INTERFACE I_UnitTest EXTENDS __SYSTEM.IQueryInterface

METHOD InitBase
VAR_INPUT
END_VAR
END_METHOD

PROPERTY Name : T_MaxString
GET
END_GET
END_PROPERTY

METHOD FINAL RunTest
END_METHOD

PROPERTY TestCompleted : BOOL
GET
END_GET
END_PROPERTY

PROPERTY TestFailed : BOOL
GET
END_GET
END_PROPERTY

END_INTERFACE

(* stored: Version 1.1.0.1, ProductVersion 3.1.4024.12
   Itf I_UnitTest: Id {4767838a-0718-44ba-96a4-9c2a6c57af2f}
   Folder Methods: Id {f66815a2-79a3-4000-9a33-2104bd81cf4b}
   Folder Properties: Id {0dcf6e56-0e3d-469a-9fcd-dd7362e9d78d}
   Method InitBase: Id {09ec4ed5-09ae-4553-8c1c-9702dbc2130b}
   Property Name: Id {d85c3f5c-1927-49ae-a32d-fca698fc6561}
   Get Get: Id {58856858-eae2-4693-9f94-3098e83eca82}
   Method RunTest: Id {e90f441b-bd22-4536-957d-3ae775f3b3a3}
   Property TestCompleted: Id {46f30332-182c-4824-9bb3-3df8be58c33f}
   Get Get: Id {63adfc7e-ea85-45ae-ad1b-548a69de2f27}
   Property TestFailed: Id {c35c2ea4-365c-4b80-b87f-9dd892be773a}
   Get Get: Id {156ac8cb-ac02-46cb-982d-9bc09bdc394e} *)
